(* IEC 61131-3 sources: plcassist-cli/packages/volt-lsp-iec/test-corpus/lenze-mid/Device/Plc Logic/Application/OEE/Local/_FirstErrorCapture, 2 files *)

(* ---- GVL_FirstErrCapture.gvl ---- *)
{attribute 'qualified_only'}
VAR_GLOBAL

//-----------------------------------------------------------------------------------------------------------------------------------------------
// O E E  I N P U T   S T R U C T U R E
//-----------------------------------------------------------------------------------------------------------------------------------------------
	asErrorCategory 	: scCategoryStruct;			// Category strings
	scFirstErrorData	: L_FECA.scErrorData;		// Data of the first error captured

	scErrorAccess : scErrorAccess;					// This structue is required using the the previous Application Template use ErrorAccess FB

 	sReasonTextPowerOn	: STRING := 'Machine switched off/on cycle';	// Text string for Mode=0 and Category=0 Power/Machine off/on cycle
//-----------------------------------------------------------------------------------------------------------------------------------------------
// L O C A L  V A R I A B L E  A N D  S T R U C T U R E
//-----------------------------------------------------------------------------------------------------------------------------------------------
	ascErrorInfo 		: ARRAY[0..GVL_ErrCapt.iErrorQty] OF  L_IE1P_ErrorInfo;			// Global strcuture for all scErrorInfo of L_IE1P_SetErrorSingle
	ascAddErrorInfo 	: ARRAY[0..GVL_ErrCapt.iErrorQty] OF  L_FECA.scErrorData_base;	// Global strcuture for all additional scErrorInfo of L_IE1P_SetErrorSingle

	scFastErrorInfo 		:  L_IE1P_ErrorInfo;		 // Global strcuture for all scErrorInfo of L_IE1P_SetErrorSingle
	scFastAddErrorInfo 		:  L_FECA.scErrorData_base;	 // Global strcuture for all additional scErrorInfo of L_IE1P_SetErrorSingle

	scOverwriteErrorInfo 		:  L_IE1P_ErrorInfo;		 // Global strcuture for one overwrite scErrorInfo of L_IE1P_SetErrorSingle
	scOverwriteAddErrorInfo 	:  L_FECA.scErrorData_base;	 // Global strcuture for one overwrite additional scErrorInfo of L_IE1P_SetErrorSingle

	xFirstErrorBit		: BOOL;
	xResetFirstError	: BOOL;

END_VAR

(* ---- FirstErrorCapture.prg ---- *)
(************************************************************************************************
*
* Program  : 	 FirstErrorCapture
*
* Summary : 	This program is used for the first error capture
*
*
* History :
*
*   Date        Author          Version    Changes
*  ------------------------------------------------------------------------------------------------------------------------------------------------------------
*
*   2023-12-21  Michael May    			1.3		Add Timer fbTonEnableDelay
*   2023-09-15  Michael May    			1.2		Insert FB L_OverwriteFirstErrCapture
*   2023-08-29  Michael May    			1.1		Use FB L_FECA.L_GetErrorTextFromFileReadArray - only
*   2023-02-24  Michael May    			1.0		Inital Version
*)

PROGRAM FirstErrorCapture
VAR

	fbFirstErrCaptureSetErrorSingle : L_FECA.L_FirstErrCaptureSetErrorSingle;		//Root cause failure detection

	fbFirstErrCapture: L_FirstFASTErrCapture;							//Root cause failure detection LEM
	fbFirstErrCaptureErrorAccess	: L_FirstErrCaptureErrorAccess;		//Root cause failure detection previous AT

	fbOverwriteFirstErrCapture: L_FECA.L_OverwriteFirstErrCapture;

	fbGetErrorTextFromFileArray :	L_GetErrorTextFromFileReadArray; 	//FB Reading Error text from file array
	xEnabledGetErrorTextfromFileArray: BOOL := TRUE;

	fbGetErrorTextFromFun : L_GetErrorTextFromFunction;					// FB Getting Error text from PLC function
	xEnabledGetErrorTextfromFun: BOOL := TRUE;

	xActivateFastErrorInput	: BOOL	:= TRUE;		// If TRUE the FAST Error Inputs are used aswell for First Error capture as second priority
	xCaptureAllReason		: BOOL	:= TRUE;		// If TRUE all active reason/error will be capture; if FALSE only severity Fault till Warning_Lock will be captured, not Warning and Information
	xCaptureOnlyFastError	: BOOL  :=TRUE;			// IF TRUE only FAST Fault severities will be captures, Warning_Lock/Warning and Information will be ignored (if FAST Warning/Information flooding the logbook)
	xCaptureStoreWarning_lock : BOOL	:= FALSE;	// If TRUE  Warning_lock priority will be stored capture like a error, If FALSE it will be handeld like a Warining or Information and can be overwritten through and error
	xPrioFromError			: BOOL	:= TRUE;		// If True Priority is taken from Error, if False Priority is taken from Category (Error or Warning/Information)

	asErrorCategoryLib 		: L_FECA.scCategoryStruct;					// 	Category strings
	xStructError	: BOOL;

	trig_NewGoodProductDetected: R_TRIG;		//TRUE if new Product/Part has been producued
	lrLastGoodPartCounter	: LREAL;			// Last Good Part Counter value
	ctuGoodPartTriggerCount	: CTU;
	xEnabledOverwrite: BOOL :=TRUE;				//Enable FirstErrCaptureOverwrite
	fbTonEnableDelay		: TON  := (PT:=T#10S);
END_VAR

VAR CONSTANT
	uiMaxError : UINT := 99;		// Max. Numbers of L_SetErrorSingleInfo fb or errors withing the whole PLC Project
END_VAR

//Assignment of scFirstErrorData := GVL_FirstErrCapture.scFirstErrorData;
xStructError := L_OEEA_Customizable_CopyStruct(pbySource:= ADR(GVL_FirstErrCapture.asErrorCategory),pbyTarget:=ADR(asErrorCategoryLib),
				uiSizeSource:=SIZEOF(GVL_FirstErrCapture.asErrorCategory),uiSizeTarget:=SIZEOF(asErrorCategoryLib));

call_FirstErrorCapture_FB();

END_PROGRAM

ACTION call_FirstErrorCapture_FB
NETWORK 0 FBD
  // // Example of Create an Trigger; if new good product is created then reset the stored First Error Capture
  // //
  ctuGoodPartTriggerCount(CU := trig_NewGoodProductDetected(CLK := (GVL_OEE_Var.scMachineData.scPartData.lrCountOK[1] = lrLastGoodPartCounter)), RESET := , PV := );
END_NETWORK
NETWORK 1 FBD
  lrLastGoodPartCounter := MOVE(GVL_OEE_Var.scMachineData.scPartData.lrCountOK[1]);
END_NETWORK
NETWORK 2 FBD
  // //*****************************************************************************************************************
  // // Call up L_FirstFastErrCapture for Root cause failure detection
  // // This funtion block is called once per PLC program, all input structure variable a global variable
  // // Logic for xResetFirstErrCapture has to be programmed/adapt, ussaly this BIT is True when the machine is back
  // // in automatic and execution and good parts has be produced
  // //******************************************************************************************************************
  GVL_FirstErrCapture.xFirstErrorBit := fbFirstErrCapture(xEnable := fbTonEnableDelay(IN := TRUE, PT := ), ascErrorInfo := GVL_FirstErrCapture.ascErrorInfo, ascAddErrorInfo := GVL_FirstErrCapture.ascAddErrorInfo, scFastErrorInfo := GVL_FirstErrCapture.scFastErrorInfo, scFastAddErrorInfo := GVL_FirstErrCapture.scFastAddErrorInfo, xActivateFastErrorInput := xActivateFastErrorInput, xCaptureAllReason := xCaptureAllReason, xCaptureOnlyFastError := xCaptureOnlyFastError, xCaptureStoreWarning_lock := xCaptureStoreWarning_lock, xPrioFromError := xPrioFromError, xResetFirstErrCapture := ((GVL_FirstErrCapture.xResetFirstError OR (trig_NewGoodProductDetected.Q AND fbFirstErrCapture.xErrorActive AND fbFirstErrCapture.xIsWarningInfo)) AND (GVL_OEE_Var.eStatus_States = eStates.Execute) AND (GVL_OEE_Var.eStatus_Modes = eModes.Production)), uiMaxError := uiMaxError, iProductionMode := GVL_OEE_Var.iProductionMode);
END_NETWORK
NETWORK 3 FBD
  fbOverwriteFirstErrCapture(xEnable := (xEnabledOverwrite AND fbTonEnableDelay.Q), scFirstErrorData := fbFirstErrCapture.scFirstErrorData, scErrorInfo := GVL_FirstErrCapture.scOverwriteErrorInfo, scAddErrorInfo := GVL_FirstErrCapture.scOverwriteAddErrorInfo, iProductionMode := GVL_OEE_Var.iProductionMode, scOutFirstErrorData => GVL_FirstErrCapture.scFirstErrorData);
END_NETWORK
NETWORK 4 FBD
  // //****************************************************************************************************************************************************
  // // Mainly used if Lenze FAST Error management (LEM)
  // // Call up L_GetErrorTextFromFileArray for getting the Error/Reasoncode Text of the active error/reason message
  // // Before using this FB the FB L_ReadErrorFromFile must be used to read the error/reson code text from the error text file into the assigned array
  // //*****************************************************************************************************************************************************
  fbGetErrorTextFromFileArray(xEnabled := (xEnabledGetErrorTextfromFileArray AND fbTonEnableDelay.Q), xErrorActive := fbFirstErrCapture.xErrorActive, xUpdateError := (fbFirstErrCapture.xUpdateError OR fbOverwriteFirstErrCapture.xUpdateError), xOnlyUserAppErrorFromFile := TRUE, scFirstErrorData := fbOverwriteFirstErrCapture.scOutFirstErrorData, iMaxNoOfSearchLoops := , asErrorText := GVL_ReadErrorFromFile.asErrorText, adwErrorID := GVL_ReadErrorFromFile.adwErrorID, scFirstErrorDataOut => GVL_FirstErrCapture.scFirstErrorData);
END_NETWORK
NETWORK 5 FBD
END_NETWORK
NETWORK 6 FBD DISABLED
  // //****************************************************************************************************************************************************
  // // Mainly used if User/Customized error management is used - not the Lenze FAST Error management
  // // Call up L_GetErrorTextFromFunction for getting the Error/Reasoncode Text of the active error/reason message
  // // This FB Receive the error text back from PLC function GetApplicationtErrorString and internal Libr. function GetFastErrorString
  // //*****************************************************************************************************************************************************
  GVL_FirstErrCapture.scFirstErrorData := fbGetErrorTextFromFun(xEnabled := xEnabledGetErrorTextfromFun, xErrorActive := fbFirstErrCapture.xErrorActive, xUpdateError := fbFirstErrCapture.xUpdateError, scFirstErrorData := fbFirstErrCapture.scFirstErrorData);
END_NETWORK
NETWORK 7 FBD
END_NETWORK
NETWORK 8 FBD DISABLED
  // //*************************************************************************************************************************************
  // // Call up L_FirstErrCaptureErrorAccess for Root cause failure detection (used with older Application Template use ErrorAccess FB)
  // // This funtion block is called once per PLC program, all input structure variable a global variable
  // // Logic for xResetFirstErrCapture has to be programmed/adapt, ussaly this BIT is True when the machine is back
  // // in automatic and execution and good parts has be produced
  // //************************************************************************************************************************************
  GVL_FirstErrCapture.xFirstErrorBit := fbFirstErrCaptureErrorAccess(xEnable := xStructError, xPrioFromError := xPrioFromError, xResetFirstErrCapture := ((GVL_FirstErrCapture.xResetFirstError OR (trig_NewGoodProductDetected.Q AND fbFirstErrCaptureErrorAccess.xErrorActive AND fbFirstErrCaptureErrorAccess.xIsWarningInfo)) AND (GVL_OEE_Var.eStatus_States = eStates.Execute) AND (GVL_OEE_Var.eStatus_Modes = eModes.Production)), scErrorAccess := GVL_FirstErrCapture.scErrorAccess, iProductionMode := GVL_OEE_Var.iProductionMode, aCategoryString := asErrorCategoryLib, scFirstErrorData => GVL_FirstErrCapture.scFirstErrorData);
END_NETWORK
END_ACTION
